Staubli VAL3: isSessionFound.pgx

program isSessionFound(string& x_sName[], num& x_nResult[])
  local string l_sString
  local bool l_bFound
  local num l_nX
  local num l_nY
  local num i
  local string l_sMessage
begin
  // look if the trajectory already exist
  call language:message(l_sString,21)
  call use:timerDialog(l_sString,0)
  l_nX=(40-len(l_sString))/2
  l_nY=5
  // read the sessino list
  call use:read(l_nX+len(l_sString),l_nY,x_sName,10,false)
  // look for the special char . and /
  if find(x_sName,".")==-1 and find(x_sName,"/")==-1 and find(x_sName,"*")==-1 and find(x_sName,"?")==-1 and find(x_sName,":")==-1 and find(x_sName,chr(34))==-1 and find(x_sName,"\")==-1
    if !use:bUseEscape
      // search inside the sSession
      for i=0 to size(sSession)-1
        if x_sName==sSession[i]
          // trajectory already exist
          call language:message(l_sString,-2)
          popUpMsg(l_sString)
          x_nResult=-1
          return
        endIf
      endFor
    else
      x_nResult=-1
    endIf
  else
    x_nResult=-1
    call language:message(l_sMessage,-3)
    l_sMessage=l_sMessage+" . / * ? : \ "+ chr(34)+" "
    popUpMsg(l_sMessage)
  endIf
end
